{attribute wpf [Container(Layout.GroupBox)]}
TYPE LayoutGroupBoxStruct EXTENDS VariousTypesStruct :
STRUCT
END_STRUCT
END_TYPE

(* stored: Version 1.1.0.1, ProductVersion 3.1.4024.9
   DUT LayoutGroupBoxStruct: Id {ac01bb8c-804e-4564-b136-a6af33b09922} *)
